Fanuc TP program (LS listing): bg_info.ls

/PROG bg_info
/ATTR
OWNER       = MNEDITOR;
CREATE      = DATE 100-11-20  TIME 09:43:21;
MODIFIED    = DATE 100-12-05  TIME 05:26:29;
LINE_COUNT = 999;
PROTECT     = READ_WRITE;
TCD:  STACK_SIZE    = 0,
      TASK_PRIORITY = 50,
      TIME_SLICE    = 0,
      BUSY_LAMP_OFF = 0,
      ABORT_REQUEST = 0,
      PAUSE_REQUEST = 0;
DEFAULT_GROUP   = 1,1,*,*,*;
CONTROL_CODE    = 00000000 00000000;
/MN
: R[30]=$SCR_GRP[1].$MCH_POS_Z;
: R[29]=$SCR_GRP[1].$MCH_POS_Y;
: R[28]=$SCR_GRP[1].$MCH_POS_X;
/POS
/END
